# EPICS autosave request: iocBoot/ioc13test/auto_positions.req
file "CARS_motor_positions.req",         P=$(P), M=m1
file "CARS_motor_positions.req",         P=$(P), M=m2
file "CARS_motor_positions.req",         P=$(P), M=m3
file "CARS_motor_positions.req",         P=$(P), M=m4
file "CARS_motor_positions.req",         P=$(P), M=m5
file "CARS_motor_positions.req",         P=$(P), M=m6
file "CARS_motor_positions.req",         P=$(P), M=m7
file "CARS_motor_positions.req",         P=$(P), M=m8
~
